SUBAPPLICATION Uebung_037 (* Spiegelabfolge V2 mit Schrittkette ENDLOS *)
  (* Standard: 61499-2 *)
  (* Version 1.0, 2023-10-23, franz *)
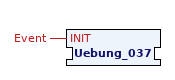
  EVENT_INPUT
    INIT;
  END_EVENT
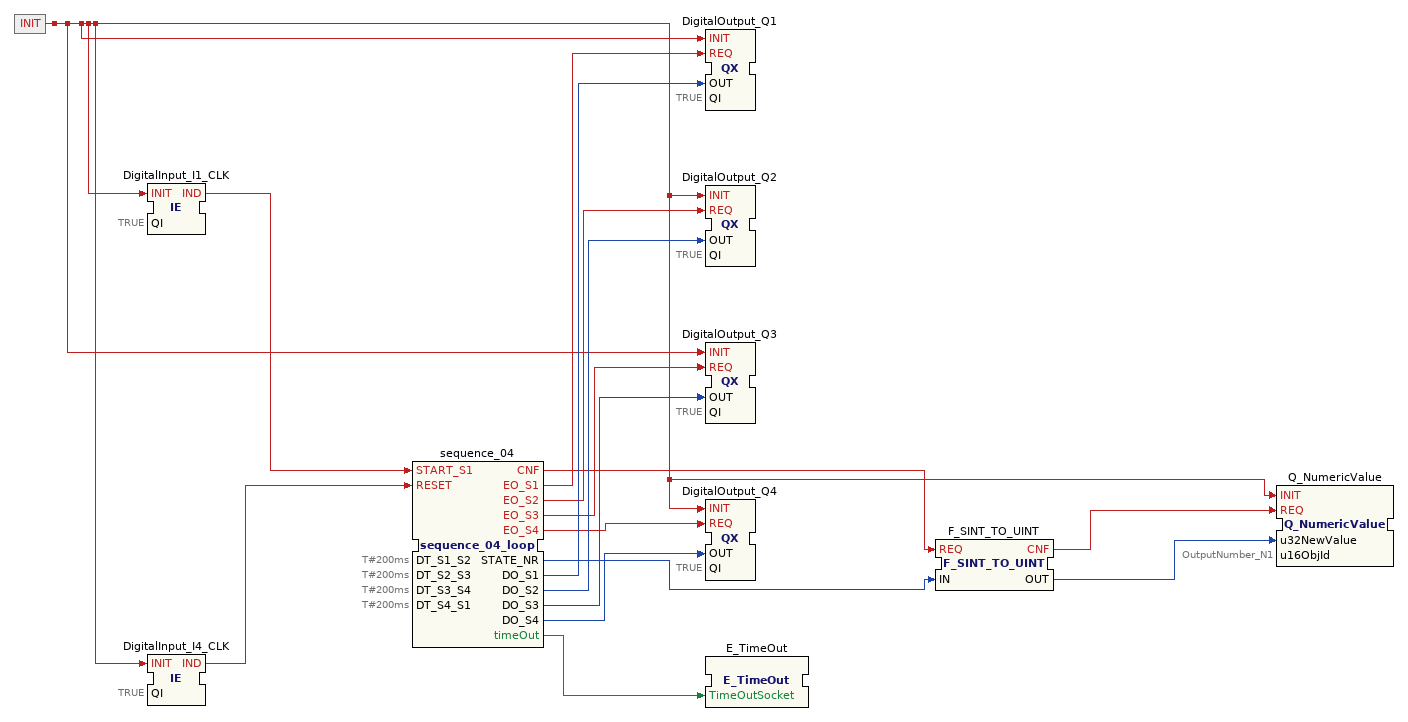
  FBS
    DigitalOutput_Q1 : QX(QI := TRUE);
    E_TimeOut : E_TimeOut;
    DigitalOutput_Q2 : QX(QI := TRUE);
    DigitalOutput_Q3 : QX(QI := TRUE);
    DigitalOutput_Q4 : QX(QI := TRUE);
    DigitalInput_I1_CLK : IE(QI := TRUE);
    DigitalInput_I4_CLK : IE(QI := TRUE);
    Q_NumericValue : Q_NumericValue(u16ObjId := OutputNumber_N1);
    F_SINT_TO_UINT : F_SINT_TO_UINT;
    sequence_04 : sequence_04_loop(DT_S1_S2 := T#200ms, DT_S2_S3 := T#200ms, DT_S3_S4 := T#200ms, DT_S4_S1 := T#200ms);
  END_FBS
  EVENT_CONNECTIONS
    INIT TO DigitalOutput_Q4.INIT;
    INIT TO DigitalOutput_Q3.INIT;
    INIT TO DigitalOutput_Q2.INIT;
    INIT TO DigitalOutput_Q1.INIT;
    INIT TO DigitalInput_I1_CLK.INIT;
    INIT TO DigitalInput_I4_CLK.INIT;
    INIT TO Q_NumericValue.INIT;
    F_SINT_TO_UINT.CNF TO Q_NumericValue.REQ;
    DigitalInput_I1_CLK.IND TO sequence_04.START_S1;
    DigitalInput_I4_CLK.IND TO sequence_04.RESET;
    sequence_04.CNF TO F_SINT_TO_UINT.REQ;
    sequence_04.EO_S1 TO DigitalOutput_Q1.REQ;
    sequence_04.EO_S2 TO DigitalOutput_Q2.REQ;
    sequence_04.EO_S3 TO DigitalOutput_Q3.REQ;
    sequence_04.EO_S4 TO DigitalOutput_Q4.REQ;
  END_CONNECTIONS
  DATA_CONNECTIONS
    F_SINT_TO_UINT.OUT TO Q_NumericValue.u32NewValue;
    sequence_04.STATE_NR TO F_SINT_TO_UINT.IN;
    sequence_04.DO_S1 TO DigitalOutput_Q1.OUT;
    sequence_04.DO_S2 TO DigitalOutput_Q2.OUT;
    sequence_04.DO_S3 TO DigitalOutput_Q3.OUT;
    sequence_04.DO_S4 TO DigitalOutput_Q4.OUT;
  END_CONNECTIONS
  ADAPTER_CONNECTIONS
    sequence_04.timeOut TO E_TimeOut.TimeOutSocket;
  END_CONNECTIONS
END_SUBAPPLICATION
